// TIA Portal V20 export
// export: Created 2026-04-11T06:02:30.3428259Z, ExportSetting WithDefaults, DisplayName Totally Integrated Automation Portal, DisplayVersion V20, DisplayName TIA Portal Openness, DisplayVersion V20, DisplayName TIA Portal Version Control Interface, DisplayVersion V20, DisplayName STEP 7 Professional, DisplayVersion V20, DisplayName STEP 7 Safety, DisplayVersion V20, DisplayName WinCC Basic/Comfort/Advanced, DisplayVersion V20, DisplayName WinCC Unified, DisplayVersion V20
TYPE "udtHMI_SoftStarter"
// stored: IsFailsafeCompliant false
   STRUCT
      iMode : Int;   // Current Mode
      iStatus { ExternalWritable := 'False'} : Int;   // Status for HMI display
      iErrorCode { ExternalWritable := 'False'} : Int;   // Error code
      bPB_ResetError : Bool;   // PB Reset errors
      bPB_On : Bool;   // PB On in manual mode
      bPB_Off : Bool;   // PB Off in manual mode
      bPBEN_ResetError { ExternalWritable := 'False'} : Bool;   // PB Reset errors enabled
      bPBEN_On { ExternalWritable := 'False'} : Bool;   // PB On enabled
      bPBEN_Off { ExternalWritable := 'False'} : Bool;   // PB Off enabled
      bOn { ExternalWritable := 'False'} : Bool;   // Soft starter on
      bSignalOnRun { ExternalWritable := 'False'} : Bool;   // Signal on/run from soft starter
      bSignalBypass { ExternalWritable := 'False'} : Bool;   // Signal bypass from soft starter
      bError { ExternalWritable := 'False'} : Bool;   // Overall Error
      bInterlock { ExternalWritable := 'False'} : Bool;   // Soft starter Interlocked
   END_STRUCT;
END_TYPE
